{attribute 'qualified_only'}
{attribute 'strict'}
TYPE E_ErrType :
(
	eFirStErr,
	eCheckBoundsErr,
	eCheckDivDint,
	eCheckDivLint,
	eCheckDivReal,
	eCheckRange,
	eCheckPointer,
	eEtherCATErr,
	eRuntimeErr,
	eLastErr
);
END_TYPE

(* stored: Version 1.1.0.1, ProductVersion 3.1.4024.4
   DUT E_ErrType: Id {18e53c82-d0cc-490b-aa11-97bc999ced61} *)
